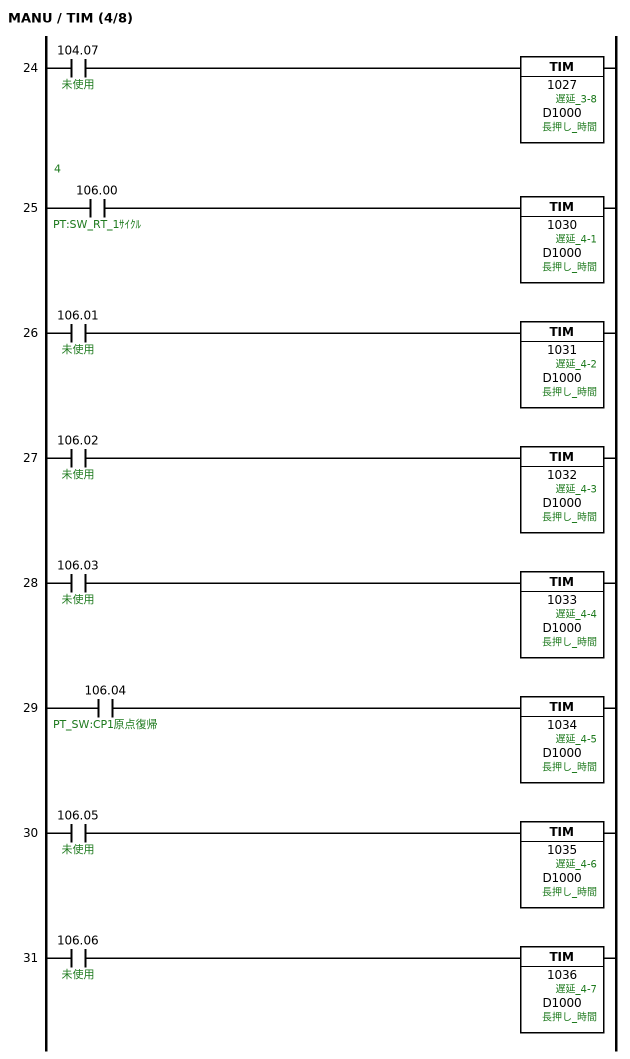
; rung 24
LD 104.07  ; 未使用
TIM 1027 D1000  ; 長押し_時間, 遅延_3-8
; rung 25: 4
LD 106.00  ; PT:SW_RT_1ｻｲｸﾙ
TIM 1030 D1000  ; 長押し_時間, 遅延_4-1
; rung 26
LD 106.01  ; 未使用
TIM 1031 D1000  ; 長押し_時間, 遅延_4-2
; rung 27
LD 106.02  ; 未使用
TIM 1032 D1000  ; 長押し_時間, 遅延_4-3
; rung 28
LD 106.03  ; 未使用
TIM 1033 D1000  ; 長押し_時間, 遅延_4-4
; rung 29
LD 106.04  ; PT_SW:CP1原点復帰
TIM 1034 D1000  ; 長押し_時間, 遅延_4-5
; rung 30
LD 106.05  ; 未使用
TIM 1035 D1000  ; 長押し_時間, 遅延_4-6
; rung 31
LD 106.06  ; 未使用
TIM 1036 D1000  ; 長押し_時間, 遅延_4-7

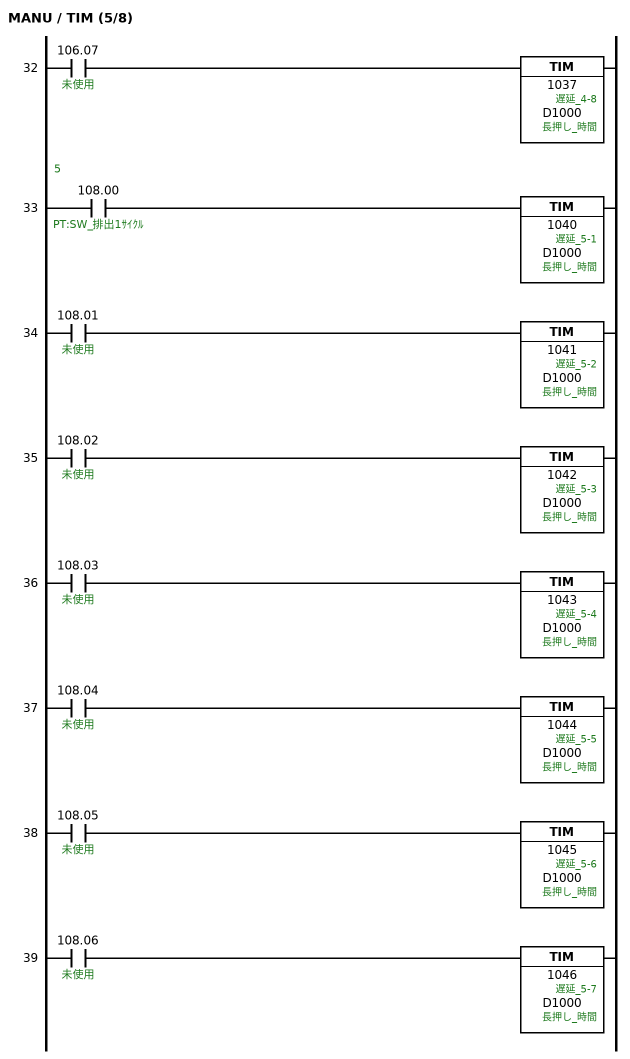
; rung 32
LD 106.07  ; 未使用
TIM 1037 D1000  ; 長押し_時間, 遅延_4-8
; rung 33: 5
LD 108.00  ; PT:SW_排出1ｻｲｸﾙ
TIM 1040 D1000  ; 長押し_時間, 遅延_5-1
; rung 34
LD 108.01  ; 未使用
TIM 1041 D1000  ; 長押し_時間, 遅延_5-2
; rung 35
LD 108.02  ; 未使用
TIM 1042 D1000  ; 長押し_時間, 遅延_5-3
; rung 36
LD 108.03  ; 未使用
TIM 1043 D1000  ; 長押し_時間, 遅延_5-4
; rung 37
LD 108.04  ; 未使用
TIM 1044 D1000  ; 長押し_時間, 遅延_5-5
; rung 38
LD 108.05  ; 未使用
TIM 1045 D1000  ; 長押し_時間, 遅延_5-6
; rung 39
LD 108.06  ; 未使用
TIM 1046 D1000  ; 長押し_時間, 遅延_5-7

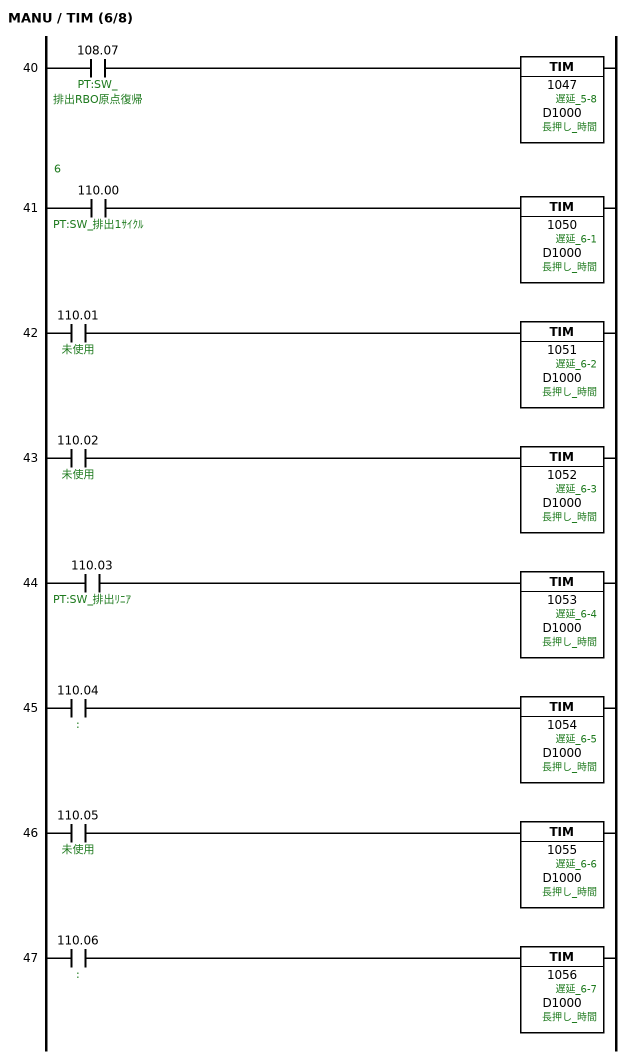
; rung 40
LD 108.07  ; PT:SW_排出RBO原点復帰
TIM 1047 D1000  ; 長押し_時間, 遅延_5-8
; rung 41: 6
LD 110.00  ; PT:SW_排出1ｻｲｸﾙ
TIM 1050 D1000  ; 長押し_時間, 遅延_6-1
; rung 42
LD 110.01  ; 未使用
TIM 1051 D1000  ; 長押し_時間, 遅延_6-2
; rung 43
LD 110.02  ; 未使用
TIM 1052 D1000  ; 長押し_時間, 遅延_6-3
; rung 44
LD 110.03  ; PT:SW_排出ﾘﾆｱ
TIM 1053 D1000  ; 長押し_時間, 遅延_6-4
; rung 45
LD 110.04  ; :
TIM 1054 D1000  ; 長押し_時間, 遅延_6-5
; rung 46
LD 110.05  ; 未使用
TIM 1055 D1000  ; 長押し_時間, 遅延_6-6
; rung 47
LD 110.06  ; :
TIM 1056 D1000  ; 長押し_時間, 遅延_6-7

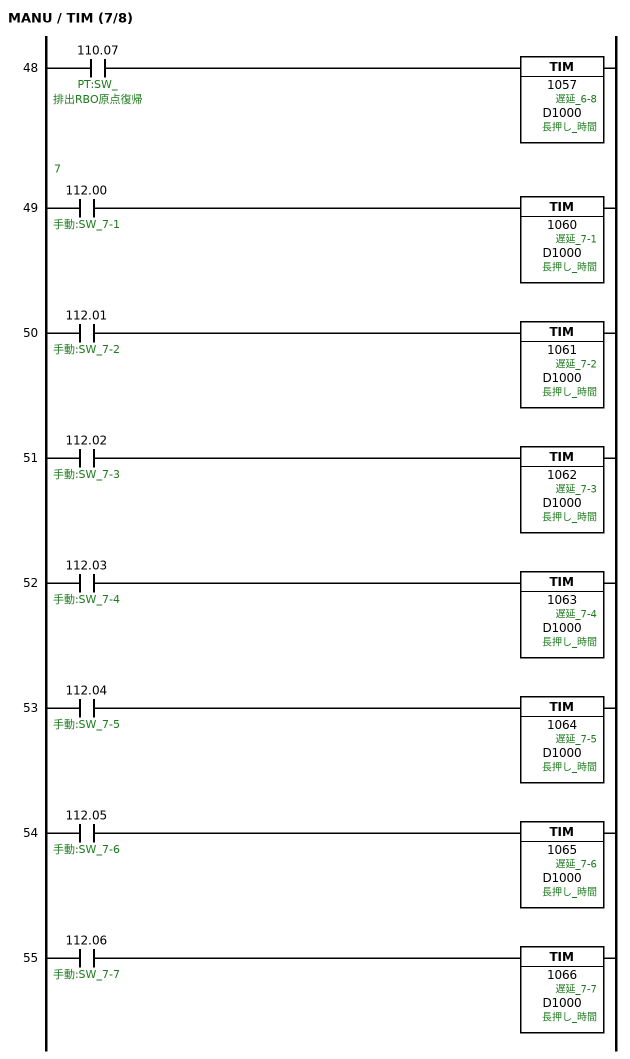
; rung 48
LD 110.07  ; PT:SW_排出RBO原点復帰
TIM 1057 D1000  ; 長押し_時間, 遅延_6-8
; rung 49: 7
LD 112.00  ; 手動:SW_7-1
TIM 1060 D1000  ; 長押し_時間, 遅延_7-1
; rung 50
LD 112.01  ; 手動:SW_7-2
TIM 1061 D1000  ; 長押し_時間, 遅延_7-2
; rung 51
LD 112.02  ; 手動:SW_7-3
TIM 1062 D1000  ; 長押し_時間, 遅延_7-3
; rung 52
LD 112.03  ; 手動:SW_7-4
TIM 1063 D1000  ; 長押し_時間, 遅延_7-4
; rung 53
LD 112.04  ; 手動:SW_7-5
TIM 1064 D1000  ; 長押し_時間, 遅延_7-5
; rung 54
LD 112.05  ; 手動:SW_7-6
TIM 1065 D1000  ; 長押し_時間, 遅延_7-6
; rung 55
LD 112.06  ; 手動:SW_7-7
TIM 1066 D1000  ; 長押し_時間, 遅延_7-7

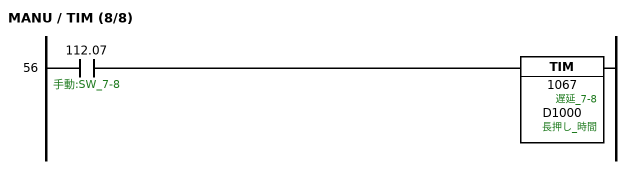
; rung 56
LD 112.07  ; 手動:SW_7-8
TIM 1067 D1000  ; 長押し_時間, 遅延_7-8

### Section MANUAL

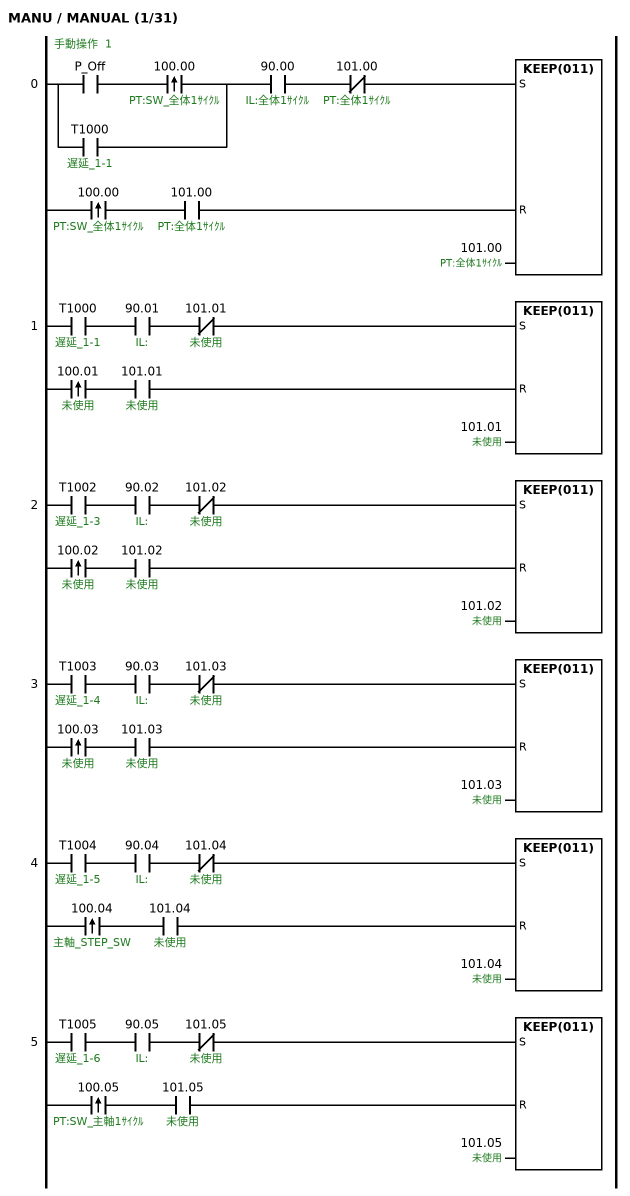
; rung 0: 手動操作  1
LD P_Off
@AND 100.00  ; PT:SW_全体1ｻｲｸﾙ
OR T1000  ; 遅延_1-1
AND 90.00  ; IL:全体1ｻｲｸﾙ
ANDNOT 101.00  ; PT:全体1ｻｲｸﾙ
@LD 100.00  ; PT:SW_全体1ｻｲｸﾙ
AND 101.00  ; PT:全体1ｻｲｸﾙ
KEEP(011) 101.00  ; PT:全体1ｻｲｸﾙ
; rung 1
LD T1000  ; 遅延_1-1
AND 90.01  ; IL:
ANDNOT 101.01  ; 未使用
@LD 100.01  ; 未使用
AND 101.01  ; 未使用
KEEP(011) 101.01  ; 未使用
; rung 2
LD T1002  ; 遅延_1-3
AND 90.02  ; IL:
ANDNOT 101.02  ; 未使用
@LD 100.02  ; 未使用
AND 101.02  ; 未使用
KEEP(011) 101.02  ; 未使用
; rung 3
LD T1003  ; 遅延_1-4
AND 90.03  ; IL:
ANDNOT 101.03  ; 未使用
@LD 100.03  ; 未使用
AND 101.03  ; 未使用
KEEP(011) 101.03  ; 未使用
; rung 4
LD T1004  ; 遅延_1-5
AND 90.04  ; IL:
ANDNOT 101.04  ; 未使用
@LD 100.04  ; 主軸_STEP_SW
AND 101.04  ; 未使用
KEEP(011) 101.04  ; 未使用
; rung 5
LD T1005  ; 遅延_1-6
AND 90.05  ; IL:
ANDNOT 101.05  ; 未使用
@LD 100.05  ; PT:SW_主軸1ｻｲｸﾙ
AND 101.05  ; 未使用
KEEP(011) 101.05  ; 未使用

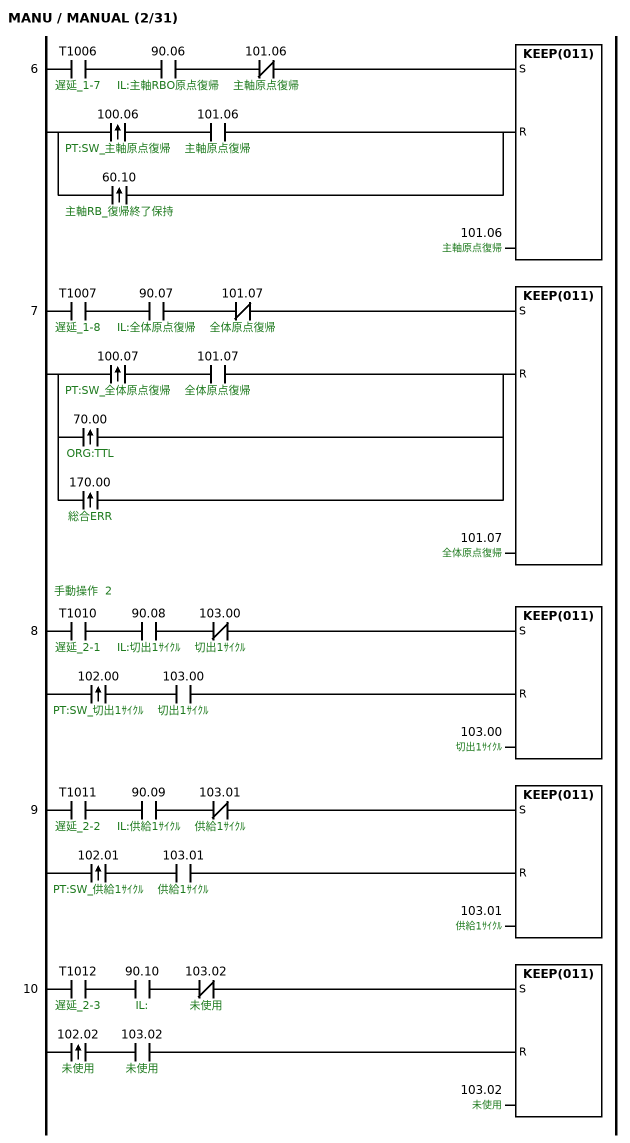
; rung 6
LD T1006  ; 遅延_1-7
AND 90.06  ; IL:主軸RBO原点復帰
ANDNOT 101.06  ; 主軸原点復帰
@LD 100.06  ; PT:SW_主軸原点復帰
AND 101.06  ; 主軸原点復帰
@OR 60.10  ; 主軸RB_復帰終了保持
KEEP(011) 101.06  ; 主軸原点復帰
; rung 7
LD T1007  ; 遅延_1-8
AND 90.07  ; IL:全体原点復帰
ANDNOT 101.07  ; 全体原点復帰
@LD 100.07  ; PT:SW_全体原点復帰
AND 101.07  ; 全体原点復帰
@OR 70.00  ; ORG:TTL
@OR 170.00  ; 総合ERR
KEEP(011) 101.07  ; 全体原点復帰
; rung 8: 手動操作  2
LD T1010  ; 遅延_2-1
AND 90.08  ; IL:切出1ｻｲｸﾙ
ANDNOT 103.00  ; 切出1ｻｲｸﾙ
@LD 102.00  ; PT:SW_切出1ｻｲｸﾙ
AND 103.00  ; 切出1ｻｲｸﾙ
KEEP(011) 103.00  ; 切出1ｻｲｸﾙ
; rung 9
LD T1011  ; 遅延_2-2
AND 90.09  ; IL:供給1ｻｲｸﾙ
ANDNOT 103.01  ; 供給1ｻｲｸﾙ
@LD 102.01  ; PT:SW_供給1ｻｲｸﾙ
AND 103.01  ; 供給1ｻｲｸﾙ
KEEP(011) 103.01  ; 供給1ｻｲｸﾙ
; rung 10
LD T1012  ; 遅延_2-3
AND 90.10  ; IL:
ANDNOT 103.02  ; 未使用
@LD 102.02  ; 未使用
AND 103.02  ; 未使用
KEEP(011) 103.02  ; 未使用

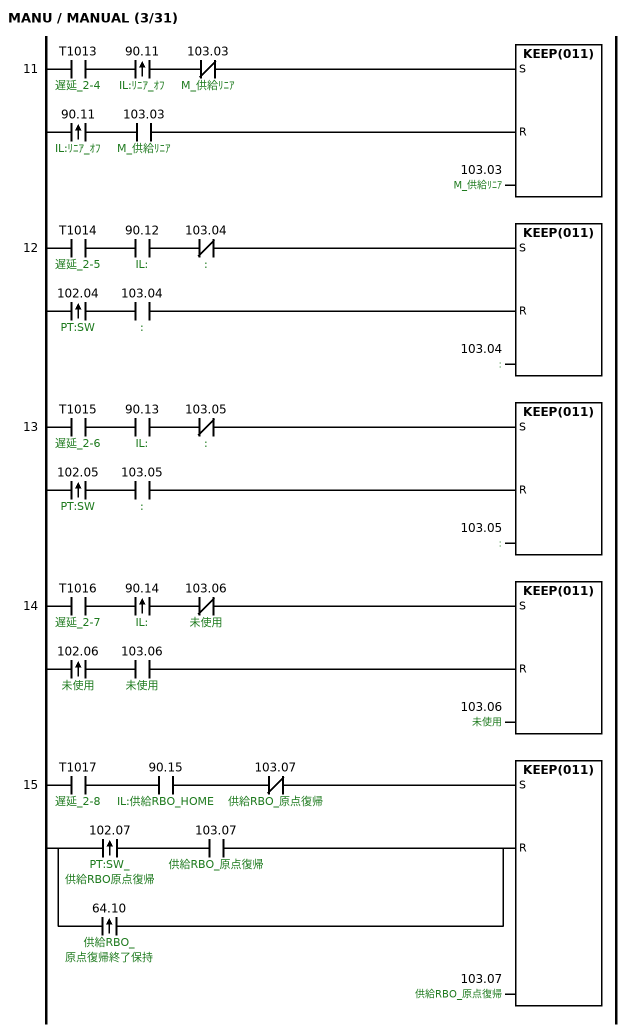
; rung 11
LD T1013  ; 遅延_2-4
@AND 90.11  ; IL:ﾘﾆｱ_ｵﾌ
ANDNOT 103.03  ; M_供給ﾘﾆｱ
@LD 90.11  ; IL:ﾘﾆｱ_ｵﾌ
AND 103.03  ; M_供給ﾘﾆｱ
KEEP(011) 103.03  ; M_供給ﾘﾆｱ
; rung 12
LD T1014  ; 遅延_2-5
AND 90.12  ; IL:
ANDNOT 103.04  ; :
@LD 102.04  ; PT:SW
AND 103.04  ; :
KEEP(011) 103.04  ; :
; rung 13
LD T1015  ; 遅延_2-6
AND 90.13  ; IL:
ANDNOT 103.05  ; :
@LD 102.05  ; PT:SW
AND 103.05  ; :
KEEP(011) 103.05  ; :
; rung 14
LD T1016  ; 遅延_2-7
@AND 90.14  ; IL:
ANDNOT 103.06  ; 未使用
@LD 102.06  ; 未使用
AND 103.06  ; 未使用
KEEP(011) 103.06  ; 未使用
; rung 15
LD T1017  ; 遅延_2-8
AND 90.15  ; IL:供給RBO_HOME
ANDNOT 103.07  ; 供給RBO_原点復帰
@LD 102.07  ; PT:SW_供給RBO原点復帰
AND 103.07  ; 供給RBO_原点復帰
@OR 64.10  ; 供給RBO_原点復帰終了保持
KEEP(011) 103.07  ; 供給RBO_原点復帰

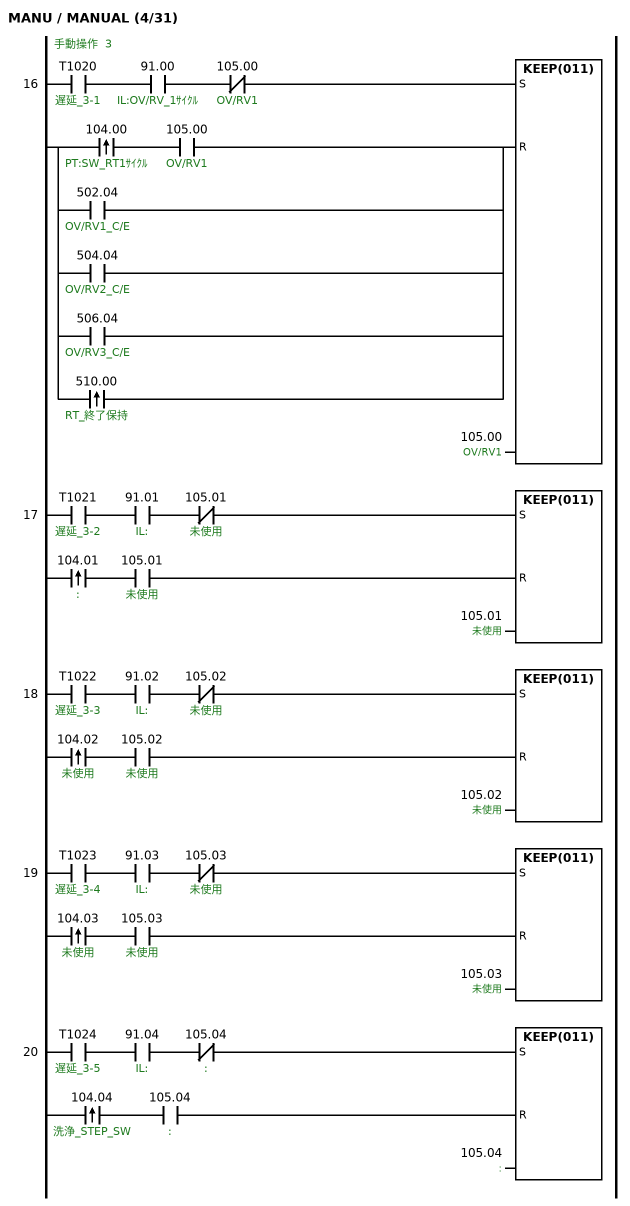
; rung 16: 手動操作  3
LD T1020  ; 遅延_3-1
AND 91.00  ; IL:OV/RV_1ｻｲｸﾙ
ANDNOT 105.00  ; OV/RV1
@LD 104.00  ; PT:SW_RT1ｻｲｸﾙ
AND 105.00  ; OV/RV1
OR 502.04  ; OV/RV1_C/E
OR 504.04  ; OV/RV2_C/E
OR 506.04  ; OV/RV3_C/E
@OR 510.00  ; RT_終了保持
KEEP(011) 105.00  ; OV/RV1
; rung 17
LD T1021  ; 遅延_3-2
AND 91.01  ; IL:
ANDNOT 105.01  ; 未使用
@LD 104.01  ; :
AND 105.01  ; 未使用
KEEP(011) 105.01  ; 未使用
; rung 18
LD T1022  ; 遅延_3-3
AND 91.02  ; IL:
ANDNOT 105.02  ; 未使用
@LD 104.02  ; 未使用
AND 105.02  ; 未使用
KEEP(011) 105.02  ; 未使用
; rung 19
LD T1023  ; 遅延_3-4
AND 91.03  ; IL:
ANDNOT 105.03  ; 未使用
@LD 104.03  ; 未使用
AND 105.03  ; 未使用
KEEP(011) 105.03  ; 未使用
; rung 20
LD T1024  ; 遅延_3-5
AND 91.04  ; IL:
ANDNOT 105.04  ; :
@LD 104.04  ; 洗浄_STEP_SW
AND 105.04  ; :
KEEP(011) 105.04  ; :

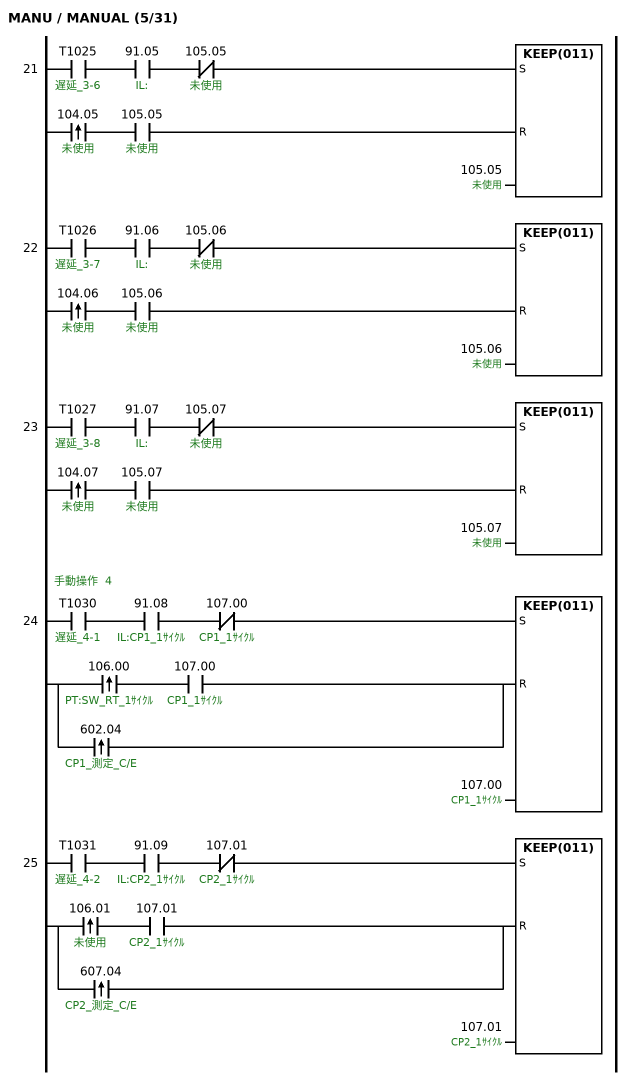
; rung 21
LD T1025  ; 遅延_3-6
AND 91.05  ; IL:
ANDNOT 105.05  ; 未使用
@LD 104.05  ; 未使用
AND 105.05  ; 未使用
KEEP(011) 105.05  ; 未使用
; rung 22
LD T1026  ; 遅延_3-7
AND 91.06  ; IL:
ANDNOT 105.06  ; 未使用
@LD 104.06  ; 未使用
AND 105.06  ; 未使用
KEEP(011) 105.06  ; 未使用
; rung 23
LD T1027  ; 遅延_3-8
AND 91.07  ; IL:
ANDNOT 105.07  ; 未使用
@LD 104.07  ; 未使用
AND 105.07  ; 未使用
KEEP(011) 105.07  ; 未使用
; rung 24: 手動操作  4
LD T1030  ; 遅延_4-1
AND 91.08  ; IL:CP1_1ｻｲｸﾙ
ANDNOT 107.00  ; CP1_1ｻｲｸﾙ
@LD 106.00  ; PT:SW_RT_1ｻｲｸﾙ
AND 107.00  ; CP1_1ｻｲｸﾙ
@OR 602.04  ; CP1_測定_C/E
KEEP(011) 107.00  ; CP1_1ｻｲｸﾙ
; rung 25
LD T1031  ; 遅延_4-2
AND 91.09  ; IL:CP2_1ｻｲｸﾙ
ANDNOT 107.01  ; CP2_1ｻｲｸﾙ
@LD 106.01  ; 未使用
AND 107.01  ; CP2_1ｻｲｸﾙ
@OR 607.04  ; CP2_測定_C/E
KEEP(011) 107.01  ; CP2_1ｻｲｸﾙ

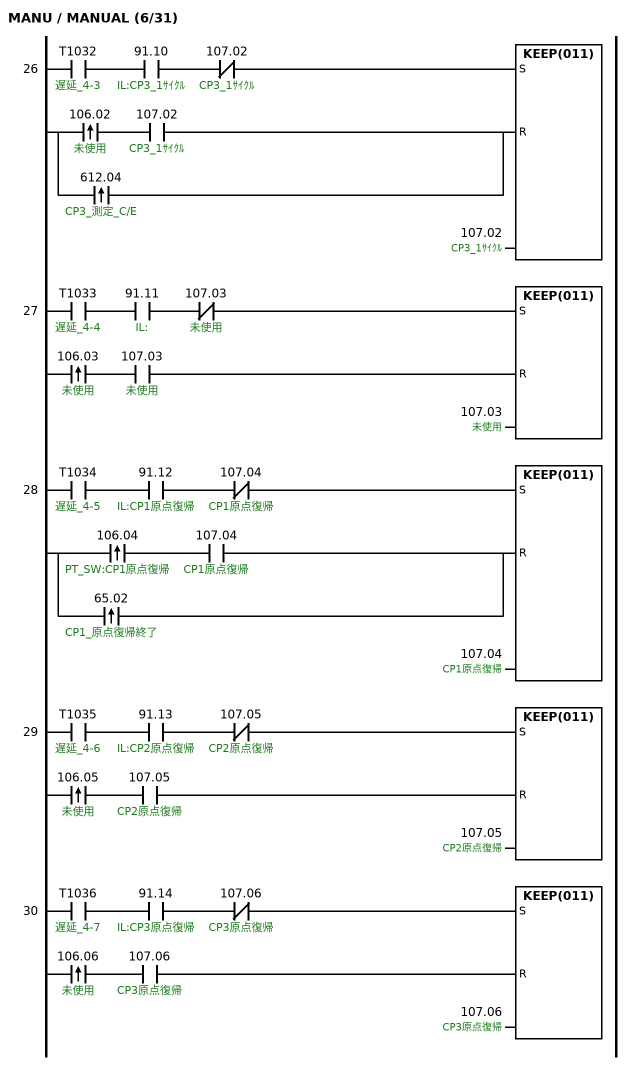
; rung 26
LD T1032  ; 遅延_4-3
AND 91.10  ; IL:CP3_1ｻｲｸﾙ
ANDNOT 107.02  ; CP3_1ｻｲｸﾙ
@LD 106.02  ; 未使用
AND 107.02  ; CP3_1ｻｲｸﾙ
@OR 612.04  ; CP3_測定_C/E
KEEP(011) 107.02  ; CP3_1ｻｲｸﾙ
; rung 27
LD T1033  ; 遅延_4-4
AND 91.11  ; IL:
ANDNOT 107.03  ; 未使用
@LD 106.03  ; 未使用
AND 107.03  ; 未使用
KEEP(011) 107.03  ; 未使用
; rung 28
LD T1034  ; 遅延_4-5
AND 91.12  ; IL:CP1原点復帰
ANDNOT 107.04  ; CP1原点復帰
@LD 106.04  ; PT_SW:CP1原点復帰
AND 107.04  ; CP1原点復帰
@OR 65.02  ; CP1_原点復帰終了
KEEP(011) 107.04  ; CP1原点復帰
; rung 29
LD T1035  ; 遅延_4-6
AND 91.13  ; IL:CP2原点復帰
ANDNOT 107.05  ; CP2原点復帰
@LD 106.05  ; 未使用
AND 107.05  ; CP2原点復帰
KEEP(011) 107.05  ; CP2原点復帰
; rung 30
LD T1036  ; 遅延_4-7
AND 91.14  ; IL:CP3原点復帰
ANDNOT 107.06  ; CP3原点復帰
@LD 106.06  ; 未使用
AND 107.06  ; CP3原点復帰
KEEP(011) 107.06  ; CP3原点復帰

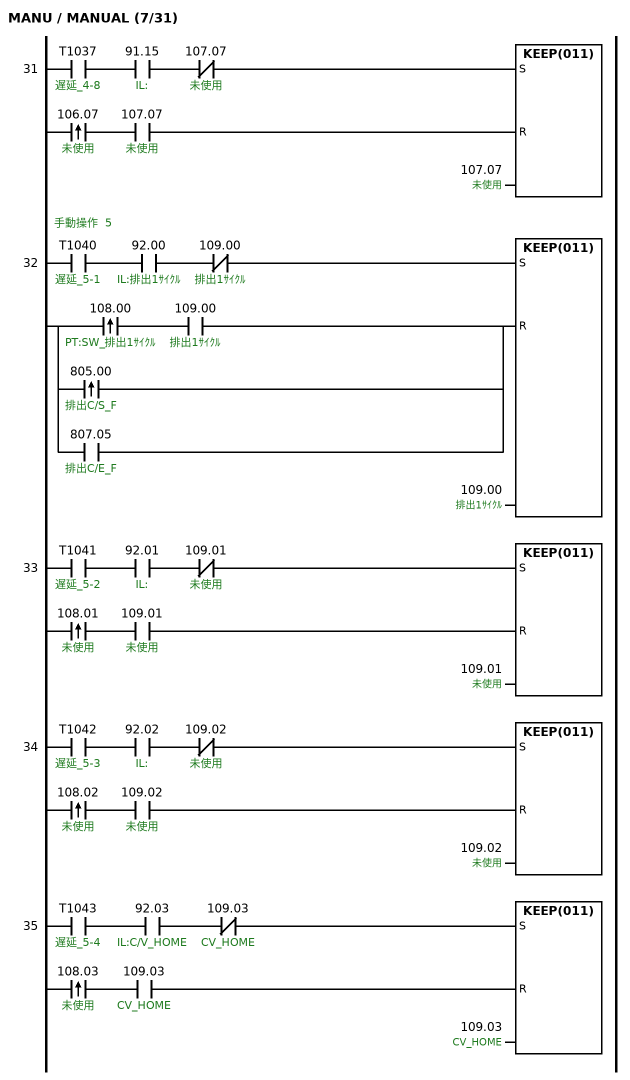
; rung 31
LD T1037  ; 遅延_4-8
AND 91.15  ; IL:
ANDNOT 107.07  ; 未使用
@LD 106.07  ; 未使用
AND 107.07  ; 未使用
KEEP(011) 107.07  ; 未使用
; rung 32: 手動操作  5
LD T1040  ; 遅延_5-1
AND 92.00  ; IL:排出1ｻｲｸﾙ
ANDNOT 109.00  ; 排出1ｻｲｸﾙ
@LD 108.00  ; PT:SW_排出1ｻｲｸﾙ
AND 109.00  ; 排出1ｻｲｸﾙ
@OR 805.00  ; 排出C/S_F
OR 807.05  ; 排出C/E_F
KEEP(011) 109.00  ; 排出1ｻｲｸﾙ
; rung 33
LD T1041  ; 遅延_5-2
AND 92.01  ; IL:
ANDNOT 109.01  ; 未使用
@LD 108.01  ; 未使用
AND 109.01  ; 未使用
KEEP(011) 109.01  ; 未使用
; rung 34
LD T1042  ; 遅延_5-3
AND 92.02  ; IL:
ANDNOT 109.02  ; 未使用
@LD 108.02  ; 未使用
AND 109.02  ; 未使用
KEEP(011) 109.02  ; 未使用
; rung 35
LD T1043  ; 遅延_5-4
AND 92.03  ; IL:C/V_HOME
ANDNOT 109.03  ; CV_HOME
@LD 108.03  ; 未使用
AND 109.03  ; CV_HOME
KEEP(011) 109.03  ; CV_HOME

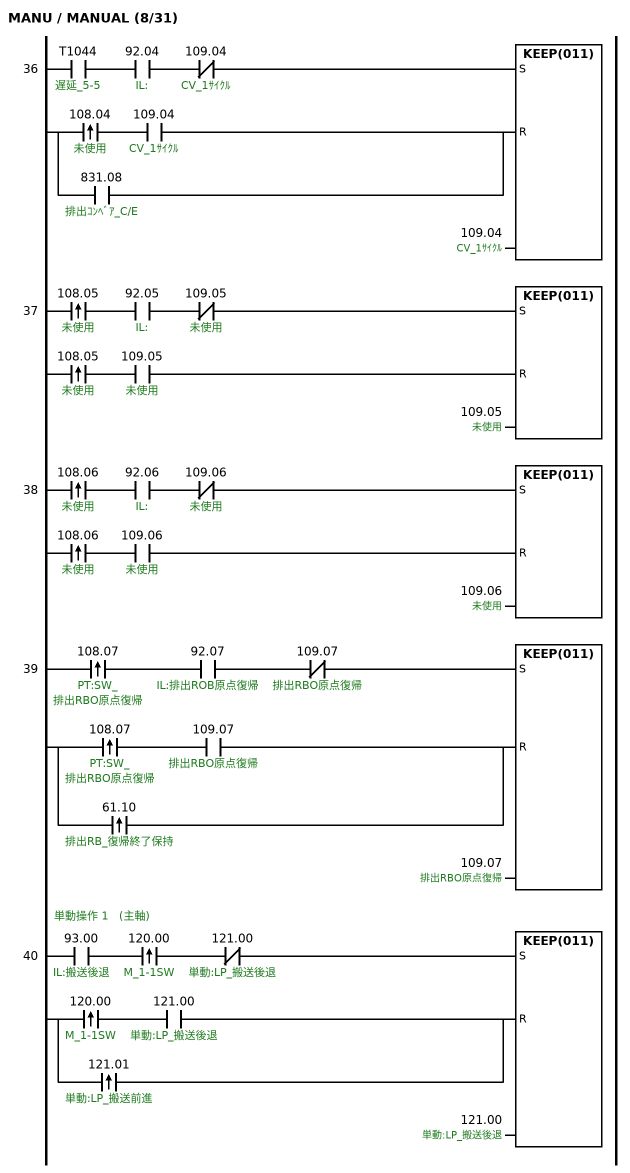
; rung 36
LD T1044  ; 遅延_5-5
AND 92.04  ; IL:
ANDNOT 109.04  ; CV_1ｻｲｸﾙ
@LD 108.04  ; 未使用
AND 109.04  ; CV_1ｻｲｸﾙ
OR 831.08  ; 排出ｺﾝﾍﾞｱ_C/E
KEEP(011) 109.04  ; CV_1ｻｲｸﾙ
; rung 37
@LD 108.05  ; 未使用
AND 92.05  ; IL:
ANDNOT 109.05  ; 未使用
@LD 108.05  ; 未使用
AND 109.05  ; 未使用
KEEP(011) 109.05  ; 未使用
; rung 38
@LD 108.06  ; 未使用
AND 92.06  ; IL:
ANDNOT 109.06  ; 未使用
@LD 108.06  ; 未使用
AND 109.06  ; 未使用
KEEP(011) 109.06  ; 未使用
; rung 39
@LD 108.07  ; PT:SW_排出RBO原点復帰
AND 92.07  ; IL:排出ROB原点復帰
ANDNOT 109.07  ; 排出RBO原点復帰
@LD 108.07  ; PT:SW_排出RBO原点復帰
AND 109.07  ; 排出RBO原点復帰
@OR 61.10  ; 排出RB_復帰終了保持
KEEP(011) 109.07  ; 排出RBO原点復帰
; rung 40: 単動操作 1   (主軸)
LD 93.00  ; IL:搬送後退
@AND 120.00  ; M_1-1SW
ANDNOT 121.00  ; 単動:LP_搬送後退
@LD 120.00  ; M_1-1SW
AND 121.00  ; 単動:LP_搬送後退
@OR 121.01  ; 単動:LP_搬送前進
KEEP(011) 121.00  ; 単動:LP_搬送後退

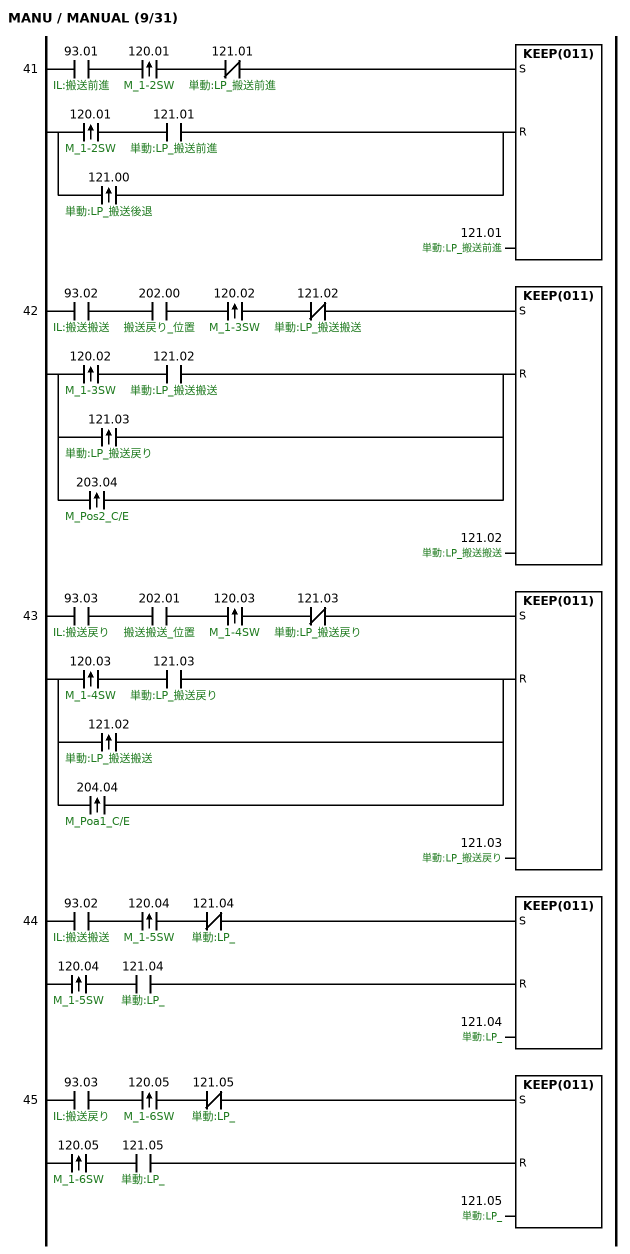
; rung 41
LD 93.01  ; IL:搬送前進
@AND 120.01  ; M_1-2SW
ANDNOT 121.01  ; 単動:LP_搬送前進
@LD 120.01  ; M_1-2SW
AND 121.01  ; 単動:LP_搬送前進
@OR 121.00  ; 単動:LP_搬送後退
KEEP(011) 121.01  ; 単動:LP_搬送前進
; rung 42
LD 93.02  ; IL:搬送搬送
AND 202.00  ; 搬送戻り_位置
@AND 120.02  ; M_1-3SW
ANDNOT 121.02  ; 単動:LP_搬送搬送
@LD 120.02  ; M_1-3SW
AND 121.02  ; 単動:LP_搬送搬送
@OR 121.03  ; 単動:LP_搬送戻り
@OR 203.04  ; M_Pos2_C/E
KEEP(011) 121.02  ; 単動:LP_搬送搬送
; rung 43
LD 93.03  ; IL:搬送戻り
AND 202.01  ; 搬送搬送_位置
@AND 120.03  ; M_1-4SW
ANDNOT 121.03  ; 単動:LP_搬送戻り
@LD 120.03  ; M_1-4SW
AND 121.03  ; 単動:LP_搬送戻り
@OR 121.02  ; 単動:LP_搬送搬送
@OR 204.04  ; M_Poa1_C/E
KEEP(011) 121.03  ; 単動:LP_搬送戻り
; rung 44
LD 93.02  ; IL:搬送搬送
@AND 120.04  ; M_1-5SW
ANDNOT 121.04  ; 単動:LP_
@LD 120.04  ; M_1-5SW
AND 121.04  ; 単動:LP_
KEEP(011) 121.04  ; 単動:LP_
; rung 45
LD 93.03  ; IL:搬送戻り
@AND 120.05  ; M_1-6SW
ANDNOT 121.05  ; 単動:LP_
@LD 120.05  ; M_1-6SW
AND 121.05  ; 単動:LP_
KEEP(011) 121.05  ; 単動:LP_

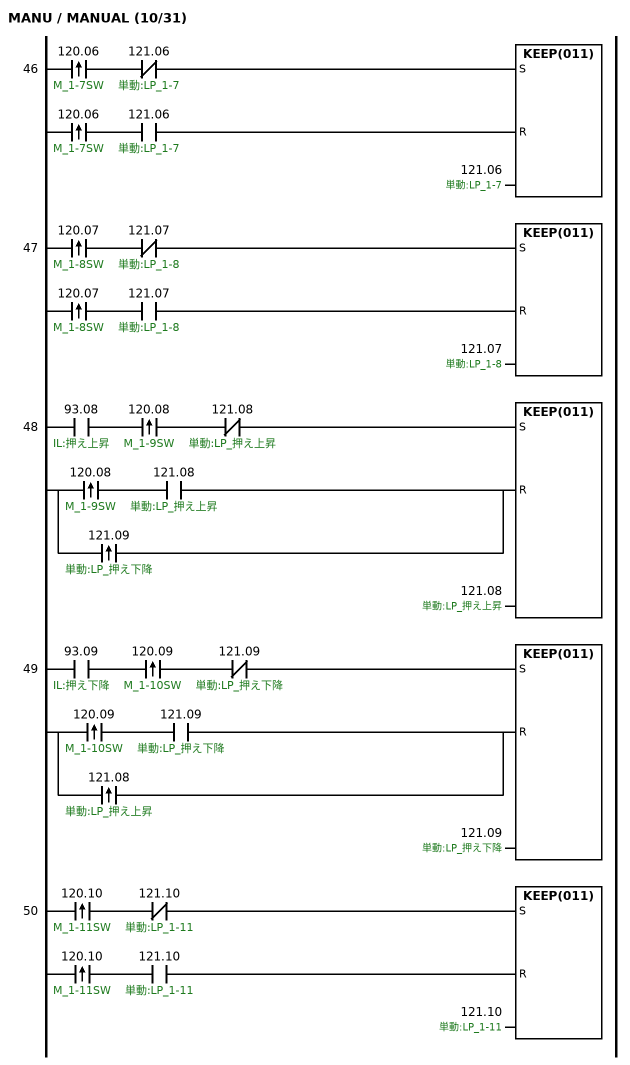
; rung 46
@LD 120.06  ; M_1-7SW
ANDNOT 121.06  ; 単動:LP_1-7
@LD 120.06  ; M_1-7SW
AND 121.06  ; 単動:LP_1-7
KEEP(011) 121.06  ; 単動:LP_1-7
; rung 47
@LD 120.07  ; M_1-8SW
ANDNOT 121.07  ; 単動:LP_1-8
@LD 120.07  ; M_1-8SW
AND 121.07  ; 単動:LP_1-8
KEEP(011) 121.07  ; 単動:LP_1-8
; rung 48
LD 93.08  ; IL:押え上昇
@AND 120.08  ; M_1-9SW
ANDNOT 121.08  ; 単動:LP_押え上昇
@LD 120.08  ; M_1-9SW
AND 121.08  ; 単動:LP_押え上昇
@OR 121.09  ; 単動:LP_押え下降
KEEP(011) 121.08  ; 単動:LP_押え上昇
; rung 49
LD 93.09  ; IL:押え下降
@AND 120.09  ; M_1-10SW
ANDNOT 121.09  ; 単動:LP_押え下降
@LD 120.09  ; M_1-10SW
AND 121.09  ; 単動:LP_押え下降
@OR 121.08  ; 単動:LP_押え上昇
KEEP(011) 121.09  ; 単動:LP_押え下降
; rung 50
@LD 120.10  ; M_1-11SW
ANDNOT 121.10  ; 単動:LP_1-11
@LD 120.10  ; M_1-11SW
AND 121.10  ; 単動:LP_1-11
KEEP(011) 121.10  ; 単動:LP_1-11

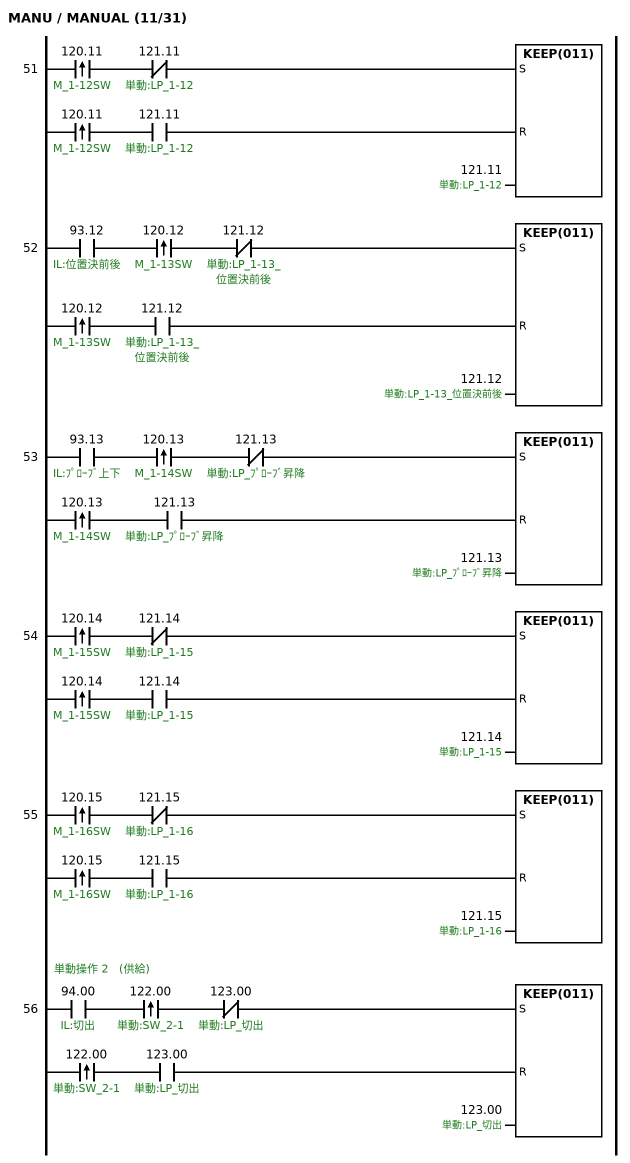
; rung 51
@LD 120.11  ; M_1-12SW
ANDNOT 121.11  ; 単動:LP_1-12
@LD 120.11  ; M_1-12SW
AND 121.11  ; 単動:LP_1-12
KEEP(011) 121.11  ; 単動:LP_1-12
; rung 52
LD 93.12  ; IL:位置決前後
@AND 120.12  ; M_1-13SW
ANDNOT 121.12  ; 単動:LP_1-13_位置決前後
@LD 120.12  ; M_1-13SW
AND 121.12  ; 単動:LP_1-13_位置決前後
KEEP(011) 121.12  ; 単動:LP_1-13_位置決前後
; rung 53
LD 93.13  ; IL:ﾌﾟﾛｰﾌﾞ上下
@AND 120.13  ; M_1-14SW
ANDNOT 121.13  ; 単動:LP_ﾌﾟﾛｰﾌﾞ昇降
@LD 120.13  ; M_1-14SW
AND 121.13  ; 単動:LP_ﾌﾟﾛｰﾌﾞ昇降
KEEP(011) 121.13  ; 単動:LP_ﾌﾟﾛｰﾌﾞ昇降
; rung 54
@LD 120.14  ; M_1-15SW
ANDNOT 121.14  ; 単動:LP_1-15
@LD 120.14  ; M_1-15SW
AND 121.14  ; 単動:LP_1-15
KEEP(011) 121.14  ; 単動:LP_1-15
; rung 55
@LD 120.15  ; M_1-16SW
ANDNOT 121.15  ; 単動:LP_1-16
@LD 120.15  ; M_1-16SW
AND 121.15  ; 単動:LP_1-16
KEEP(011) 121.15  ; 単動:LP_1-16
; rung 56: 単動操作 2   (供給)
LD 94.00  ; IL:切出
@AND 122.00  ; 単動:SW_2-1
ANDNOT 123.00  ; 単動:LP_切出
@LD 122.00  ; 単動:SW_2-1
AND 123.00  ; 単動:LP_切出
KEEP(011) 123.00  ; 単動:LP_切出

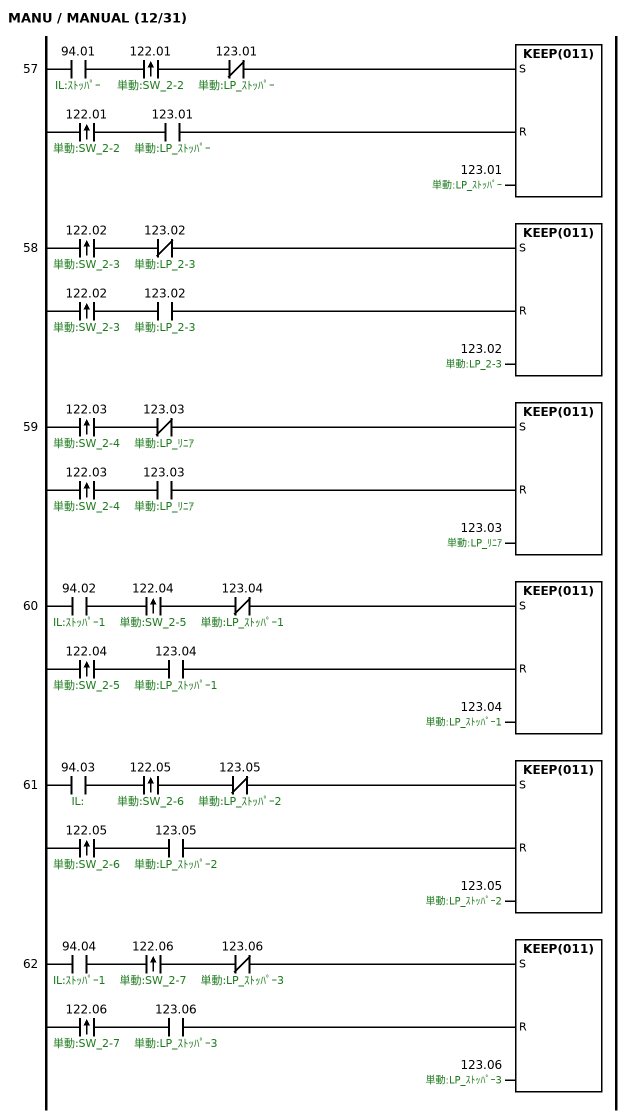
; rung 57
LD 94.01  ; IL:ｽﾄｯﾊﾟｰ
@AND 122.01  ; 単動:SW_2-2
ANDNOT 123.01  ; 単動:LP_ｽﾄｯﾊﾟｰ
@LD 122.01  ; 単動:SW_2-2
AND 123.01  ; 単動:LP_ｽﾄｯﾊﾟｰ
KEEP(011) 123.01  ; 単動:LP_ｽﾄｯﾊﾟｰ
; rung 58
@LD 122.02  ; 単動:SW_2-3
ANDNOT 123.02  ; 単動:LP_2-3
@LD 122.02  ; 単動:SW_2-3
AND 123.02  ; 単動:LP_2-3
KEEP(011) 123.02  ; 単動:LP_2-3
; rung 59
@LD 122.03  ; 単動:SW_2-4
ANDNOT 123.03  ; 単動:LP_ﾘﾆｱ
@LD 122.03  ; 単動:SW_2-4
AND 123.03  ; 単動:LP_ﾘﾆｱ
KEEP(011) 123.03  ; 単動:LP_ﾘﾆｱ
; rung 60
LD 94.02  ; IL:ｽﾄｯﾊﾟｰ1
@AND 122.04  ; 単動:SW_2-5
ANDNOT 123.04  ; 単動:LP_ｽﾄｯﾊﾟｰ1
@LD 122.04  ; 単動:SW_2-5
AND 123.04  ; 単動:LP_ｽﾄｯﾊﾟｰ1
KEEP(011) 123.04  ; 単動:LP_ｽﾄｯﾊﾟｰ1
; rung 61
LD 94.03  ; IL:
@AND 122.05  ; 単動:SW_2-6
ANDNOT 123.05  ; 単動:LP_ｽﾄｯﾊﾟｰ2
@LD 122.05  ; 単動:SW_2-6
AND 123.05  ; 単動:LP_ｽﾄｯﾊﾟｰ2
KEEP(011) 123.05  ; 単動:LP_ｽﾄｯﾊﾟｰ2
; rung 62
LD 94.04  ; IL:ｽﾄｯﾊﾟｰ1
@AND 122.06  ; 単動:SW_2-7
ANDNOT 123.06  ; 単動:LP_ｽﾄｯﾊﾟｰ3
@LD 122.06  ; 単動:SW_2-7
AND 123.06  ; 単動:LP_ｽﾄｯﾊﾟｰ3
KEEP(011) 123.06  ; 単動:LP_ｽﾄｯﾊﾟｰ3

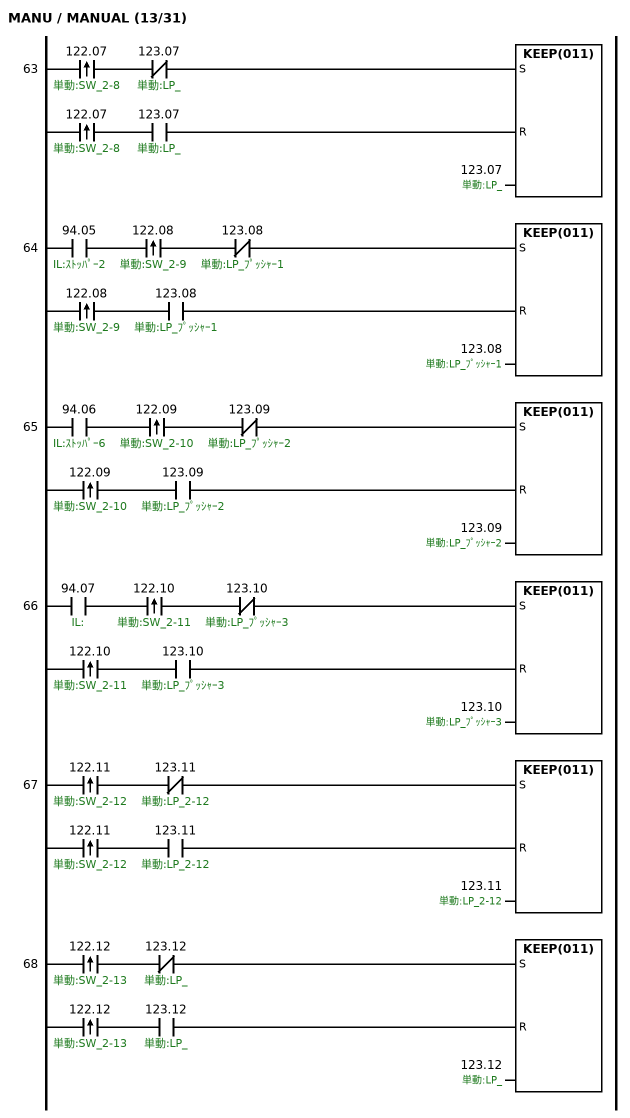
; rung 63
@LD 122.07  ; 単動:SW_2-8
ANDNOT 123.07  ; 単動:LP_
@LD 122.07  ; 単動:SW_2-8
AND 123.07  ; 単動:LP_
KEEP(011) 123.07  ; 単動:LP_
; rung 64
LD 94.05  ; IL:ｽﾄｯﾊﾟｰ2
@AND 122.08  ; 単動:SW_2-9
ANDNOT 123.08  ; 単動:LP_ﾌﾟｯｼｬｰ1
@LD 122.08  ; 単動:SW_2-9
AND 123.08  ; 単動:LP_ﾌﾟｯｼｬｰ1
KEEP(011) 123.08  ; 単動:LP_ﾌﾟｯｼｬｰ1
; rung 65
LD 94.06  ; IL:ｽﾄｯﾊﾟｰ6
@AND 122.09  ; 単動:SW_2-10
ANDNOT 123.09  ; 単動:LP_ﾌﾟｯｼｬｰ2
@LD 122.09  ; 単動:SW_2-10
AND 123.09  ; 単動:LP_ﾌﾟｯｼｬｰ2
KEEP(011) 123.09  ; 単動:LP_ﾌﾟｯｼｬｰ2
; rung 66
LD 94.07  ; IL:
@AND 122.10  ; 単動:SW_2-11
ANDNOT 123.10  ; 単動:LP_ﾌﾟｯｼｬｰ3
@LD 122.10  ; 単動:SW_2-11
AND 123.10  ; 単動:LP_ﾌﾟｯｼｬｰ3
KEEP(011) 123.10  ; 単動:LP_ﾌﾟｯｼｬｰ3
; rung 67
@LD 122.11  ; 単動:SW_2-12
ANDNOT 123.11  ; 単動:LP_2-12
@LD 122.11  ; 単動:SW_2-12
AND 123.11  ; 単動:LP_2-12
KEEP(011) 123.11  ; 単動:LP_2-12
; rung 68
@LD 122.12  ; 単動:SW_2-13
ANDNOT 123.12  ; 単動:LP_
@LD 122.12  ; 単動:SW_2-13
AND 123.12  ; 単動:LP_
KEEP(011) 123.12  ; 単動:LP_

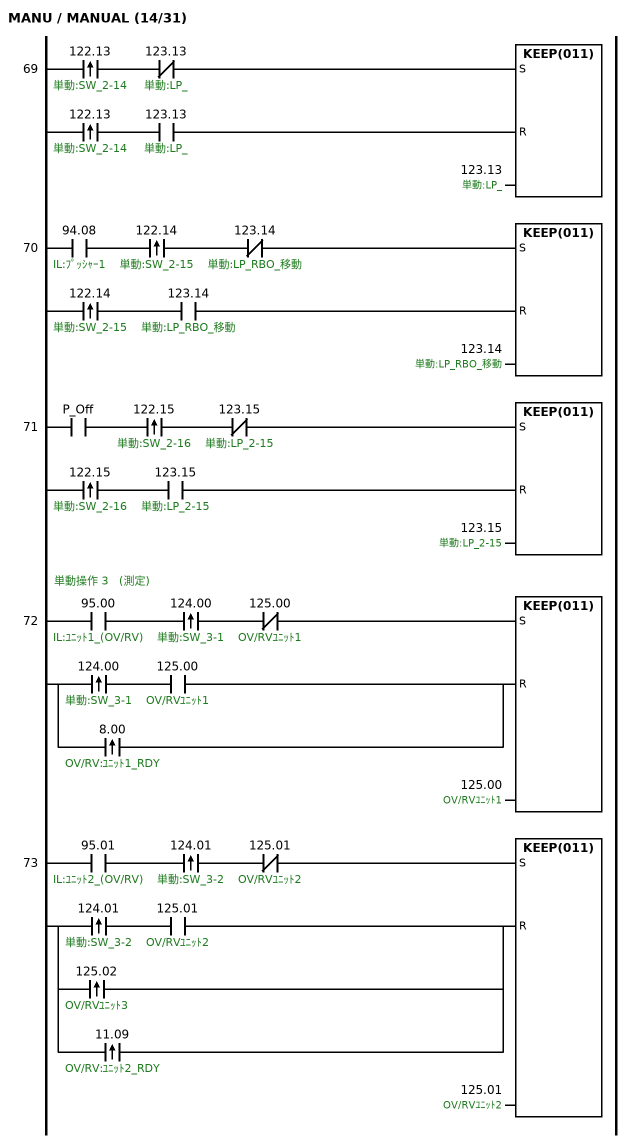
; rung 69
@LD 122.13  ; 単動:SW_2-14
ANDNOT 123.13  ; 単動:LP_
@LD 122.13  ; 単動:SW_2-14
AND 123.13  ; 単動:LP_
KEEP(011) 123.13  ; 単動:LP_
; rung 70
LD 94.08  ; IL:ﾌﾟｯｼｬｰ1
@AND 122.14  ; 単動:SW_2-15
ANDNOT 123.14  ; 単動:LP_RBO_移動
@LD 122.14  ; 単動:SW_2-15
AND 123.14  ; 単動:LP_RBO_移動
KEEP(011) 123.14  ; 単動:LP_RBO_移動
; rung 71
LD P_Off
@AND 122.15  ; 単動:SW_2-16
ANDNOT 123.15  ; 単動:LP_2-15
@LD 122.15  ; 単動:SW_2-16
AND 123.15  ; 単動:LP_2-15
KEEP(011) 123.15  ; 単動:LP_2-15
; rung 72: 単動操作 3   (測定)
LD 95.00  ; IL:ﾕﾆｯﾄ1_(OV/RV)
@AND 124.00  ; 単動:SW_3-1
ANDNOT 125.00  ; OV/RVﾕﾆｯﾄ1
@LD 124.00  ; 単動:SW_3-1
AND 125.00  ; OV/RVﾕﾆｯﾄ1
@OR 8.00  ; OV/RV:ﾕﾆｯﾄ1_RDY
KEEP(011) 125.00  ; OV/RVﾕﾆｯﾄ1
; rung 73
LD 95.01  ; IL:ﾕﾆｯﾄ2_(OV/RV)
@AND 124.01  ; 単動:SW_3-2
ANDNOT 125.01  ; OV/RVﾕﾆｯﾄ2
@LD 124.01  ; 単動:SW_3-2
AND 125.01  ; OV/RVﾕﾆｯﾄ2
@OR 125.02  ; OV/RVﾕﾆｯﾄ3
@OR 11.09  ; OV/RV:ﾕﾆｯﾄ2_RDY
KEEP(011) 125.01  ; OV/RVﾕﾆｯﾄ2

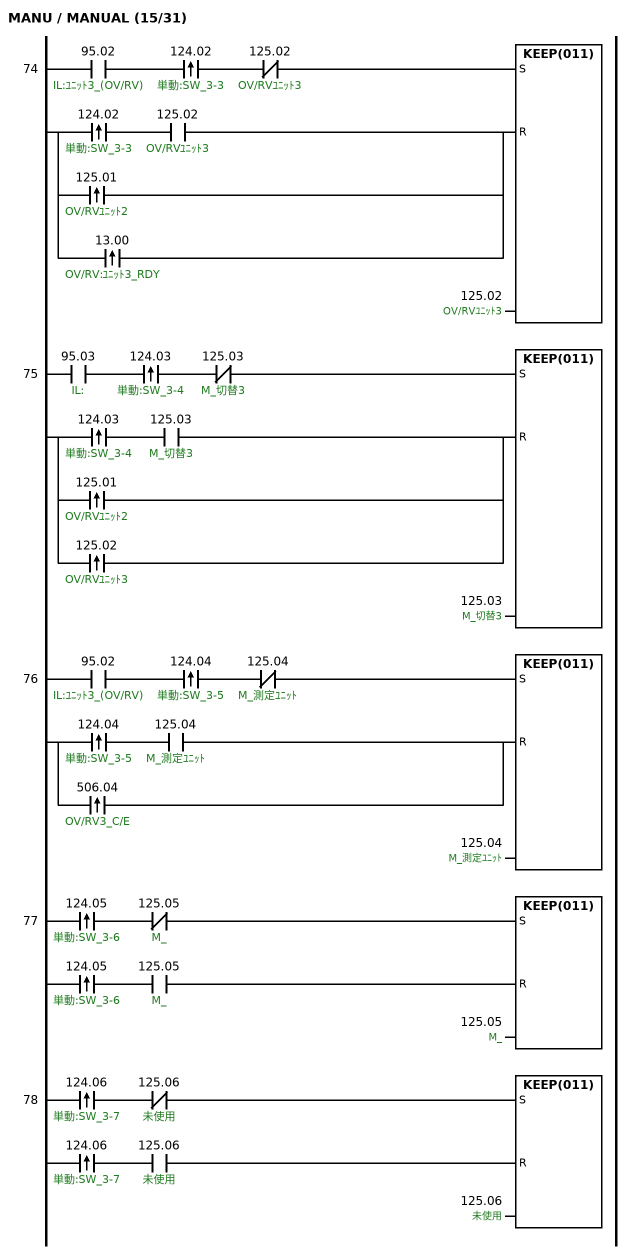
; rung 74
LD 95.02  ; IL:ﾕﾆｯﾄ3_(OV/RV)
@AND 124.02  ; 単動:SW_3-3
ANDNOT 125.02  ; OV/RVﾕﾆｯﾄ3
@LD 124.02  ; 単動:SW_3-3
AND 125.02  ; OV/RVﾕﾆｯﾄ3
@OR 125.01  ; OV/RVﾕﾆｯﾄ2
@OR 13.00  ; OV/RV:ﾕﾆｯﾄ3_RDY
KEEP(011) 125.02  ; OV/RVﾕﾆｯﾄ3
; rung 75
LD 95.03  ; IL:
@AND 124.03  ; 単動:SW_3-4
ANDNOT 125.03  ; M_切替3
@LD 124.03  ; 単動:SW_3-4
AND 125.03  ; M_切替3
@OR 125.01  ; OV/RVﾕﾆｯﾄ2
@OR 125.02  ; OV/RVﾕﾆｯﾄ3
KEEP(011) 125.03  ; M_切替3
; rung 76
LD 95.02  ; IL:ﾕﾆｯﾄ3_(OV/RV)
@AND 124.04  ; 単動:SW_3-5
ANDNOT 125.04  ; M_測定ﾕﾆｯﾄ
@LD 124.04  ; 単動:SW_3-5
AND 125.04  ; M_測定ﾕﾆｯﾄ
@OR 506.04  ; OV/RV3_C/E
KEEP(011) 125.04  ; M_測定ﾕﾆｯﾄ
; rung 77
@LD 124.05  ; 単動:SW_3-6
ANDNOT 125.05  ; M_
@LD 124.05  ; 単動:SW_3-6
AND 125.05  ; M_
KEEP(011) 125.05  ; M_
; rung 78
@LD 124.06  ; 単動:SW_3-7
ANDNOT 125.06  ; 未使用
@LD 124.06  ; 単動:SW_3-7
AND 125.06  ; 未使用
KEEP(011) 125.06  ; 未使用

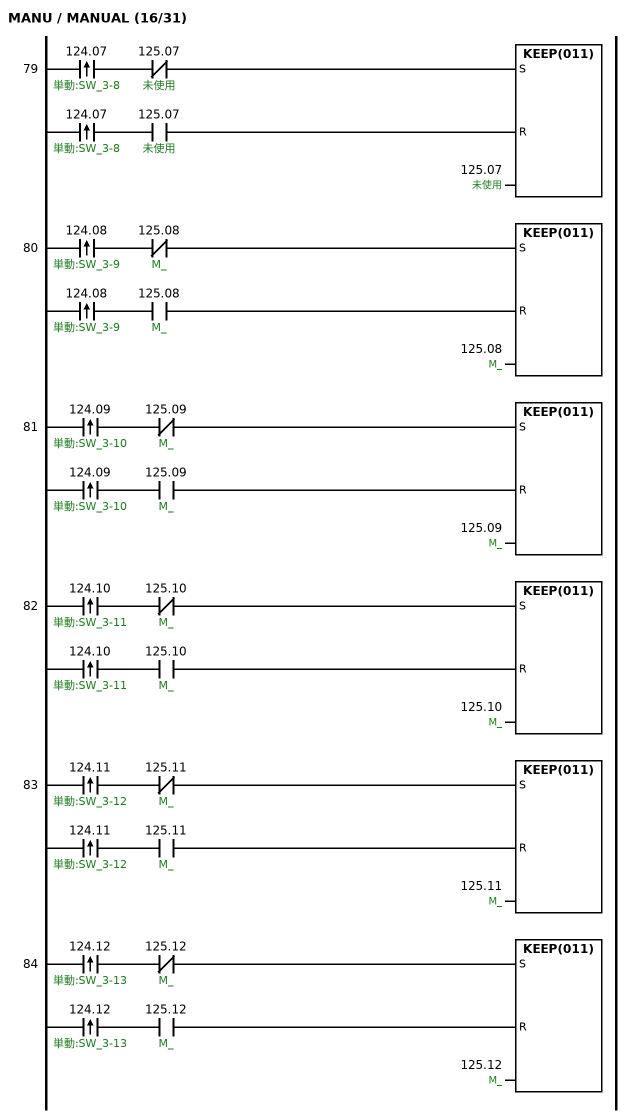
; rung 79
@LD 124.07  ; 単動:SW_3-8
ANDNOT 125.07  ; 未使用
@LD 124.07  ; 単動:SW_3-8
AND 125.07  ; 未使用
KEEP(011) 125.07  ; 未使用
; rung 80
@LD 124.08  ; 単動:SW_3-9
ANDNOT 125.08  ; M_
@LD 124.08  ; 単動:SW_3-9
AND 125.08  ; M_
KEEP(011) 125.08  ; M_
; rung 81
@LD 124.09  ; 単動:SW_3-10
ANDNOT 125.09  ; M_
@LD 124.09  ; 単動:SW_3-10
AND 125.09  ; M_
KEEP(011) 125.09  ; M_
; rung 82
@LD 124.10  ; 単動:SW_3-11
ANDNOT 125.10  ; M_
@LD 124.10  ; 単動:SW_3-11
AND 125.10  ; M_
KEEP(011) 125.10  ; M_
; rung 83
@LD 124.11  ; 単動:SW_3-12
ANDNOT 125.11  ; M_
@LD 124.11  ; 単動:SW_3-12
AND 125.11  ; M_
KEEP(011) 125.11  ; M_
; rung 84
@LD 124.12  ; 単動:SW_3-13
ANDNOT 125.12  ; M_
@LD 124.12  ; 単動:SW_3-13
AND 125.12  ; M_
KEEP(011) 125.12  ; M_

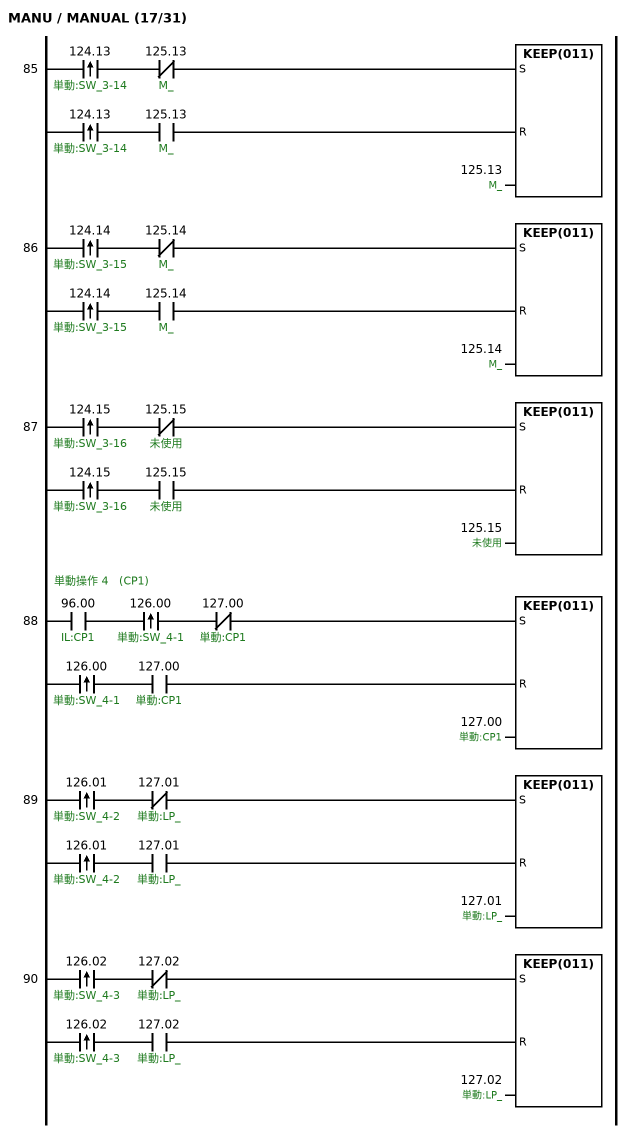
; rung 85
@LD 124.13  ; 単動:SW_3-14
ANDNOT 125.13  ; M_
@LD 124.13  ; 単動:SW_3-14
AND 125.13  ; M_
KEEP(011) 125.13  ; M_
; rung 86
@LD 124.14  ; 単動:SW_3-15
ANDNOT 125.14  ; M_
@LD 124.14  ; 単動:SW_3-15
AND 125.14  ; M_
KEEP(011) 125.14  ; M_
; rung 87
@LD 124.15  ; 単動:SW_3-16
ANDNOT 125.15  ; 未使用
@LD 124.15  ; 単動:SW_3-16
AND 125.15  ; 未使用
KEEP(011) 125.15  ; 未使用
; rung 88: 単動操作 4   (CP1)
LD 96.00  ; IL:CP1
@AND 126.00  ; 単動:SW_4-1
ANDNOT 127.00  ; 単動:CP1
@LD 126.00  ; 単動:SW_4-1
AND 127.00  ; 単動:CP1
KEEP(011) 127.00  ; 単動:CP1
; rung 89
@LD 126.01  ; 単動:SW_4-2
ANDNOT 127.01  ; 単動:LP_
@LD 126.01  ; 単動:SW_4-2
AND 127.01  ; 単動:LP_
KEEP(011) 127.01  ; 単動:LP_
; rung 90
@LD 126.02  ; 単動:SW_4-3
ANDNOT 127.02  ; 単動:LP_
@LD 126.02  ; 単動:SW_4-3
AND 127.02  ; 単動:LP_
KEEP(011) 127.02  ; 単動:LP_

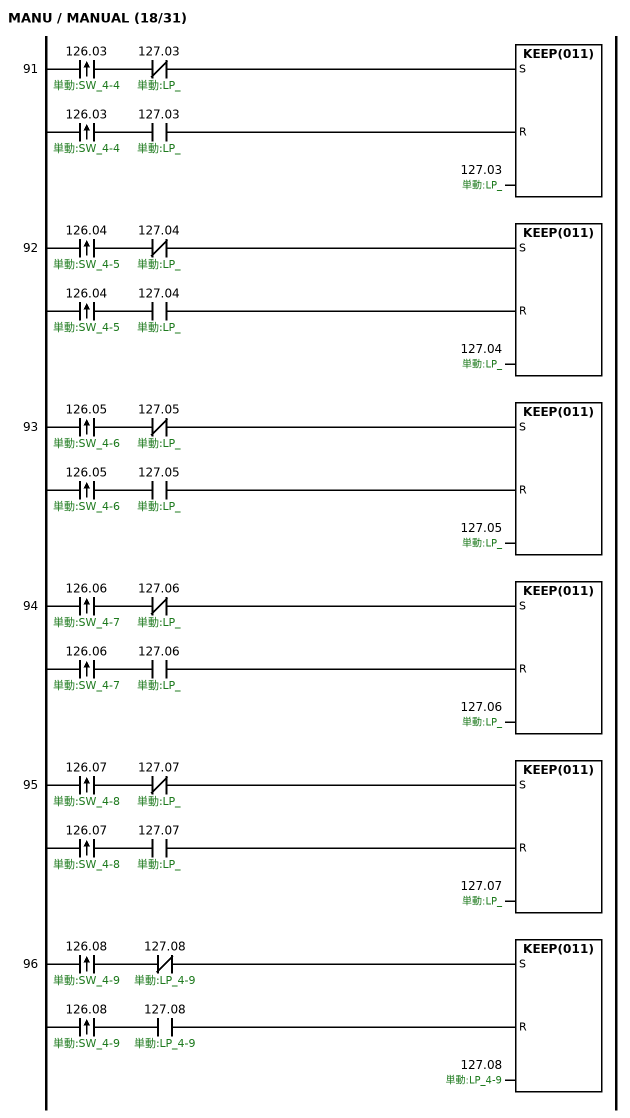
; rung 91
@LD 126.03  ; 単動:SW_4-4
ANDNOT 127.03  ; 単動:LP_
@LD 126.03  ; 単動:SW_4-4
AND 127.03  ; 単動:LP_
KEEP(011) 127.03  ; 単動:LP_
; rung 92
@LD 126.04  ; 単動:SW_4-5
ANDNOT 127.04  ; 単動:LP_
@LD 126.04  ; 単動:SW_4-5
AND 127.04  ; 単動:LP_
KEEP(011) 127.04  ; 単動:LP_
; rung 93
@LD 126.05  ; 単動:SW_4-6
ANDNOT 127.05  ; 単動:LP_
@LD 126.05  ; 単動:SW_4-6
AND 127.05  ; 単動:LP_
KEEP(011) 127.05  ; 単動:LP_
; rung 94
@LD 126.06  ; 単動:SW_4-7
ANDNOT 127.06  ; 単動:LP_
@LD 126.06  ; 単動:SW_4-7
AND 127.06  ; 単動:LP_
KEEP(011) 127.06  ; 単動:LP_
; rung 95
@LD 126.07  ; 単動:SW_4-8
ANDNOT 127.07  ; 単動:LP_
@LD 126.07  ; 単動:SW_4-8
AND 127.07  ; 単動:LP_
KEEP(011) 127.07  ; 単動:LP_
; rung 96
@LD 126.08  ; 単動:SW_4-9
ANDNOT 127.08  ; 単動:LP_4-9
@LD 126.08  ; 単動:SW_4-9
AND 127.08  ; 単動:LP_4-9
KEEP(011) 127.08  ; 単動:LP_4-9

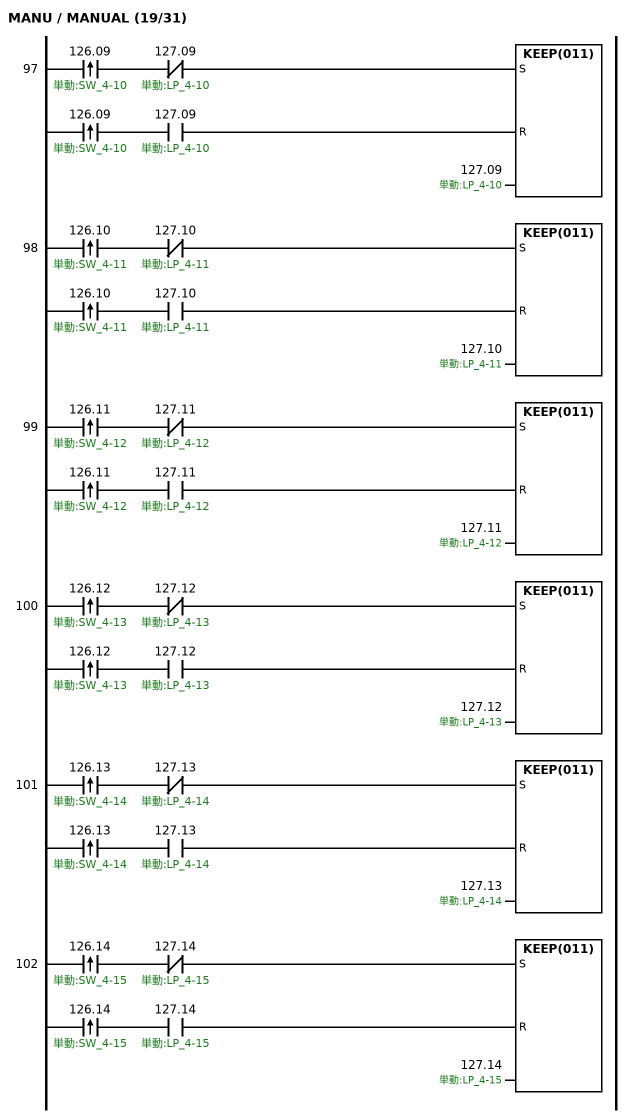
; rung 97
@LD 126.09  ; 単動:SW_4-10
ANDNOT 127.09  ; 単動:LP_4-10
@LD 126.09  ; 単動:SW_4-10
AND 127.09  ; 単動:LP_4-10
KEEP(011) 127.09  ; 単動:LP_4-10
; rung 98
@LD 126.10  ; 単動:SW_4-11
ANDNOT 127.10  ; 単動:LP_4-11
@LD 126.10  ; 単動:SW_4-11
AND 127.10  ; 単動:LP_4-11
KEEP(011) 127.10  ; 単動:LP_4-11
; rung 99
@LD 126.11  ; 単動:SW_4-12
ANDNOT 127.11  ; 単動:LP_4-12
@LD 126.11  ; 単動:SW_4-12
AND 127.11  ; 単動:LP_4-12
KEEP(011) 127.11  ; 単動:LP_4-12
; rung 100
@LD 126.12  ; 単動:SW_4-13
ANDNOT 127.12  ; 単動:LP_4-13
@LD 126.12  ; 単動:SW_4-13
AND 127.12  ; 単動:LP_4-13
KEEP(011) 127.12  ; 単動:LP_4-13
; rung 101
@LD 126.13  ; 単動:SW_4-14
ANDNOT 127.13  ; 単動:LP_4-14
@LD 126.13  ; 単動:SW_4-14
AND 127.13  ; 単動:LP_4-14
KEEP(011) 127.13  ; 単動:LP_4-14
; rung 102
@LD 126.14  ; 単動:SW_4-15
ANDNOT 127.14  ; 単動:LP_4-15
@LD 126.14  ; 単動:SW_4-15
AND 127.14  ; 単動:LP_4-15
KEEP(011) 127.14  ; 単動:LP_4-15

